ABB RobotStudio station: RoboX0_20211129-155304.rsstn

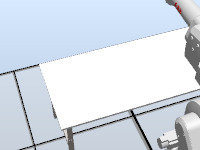
Station RoboX0 (saved by RobotStudio 21.3.9648.0)
Controller IRB1600_10_145, task T_ROB1: task frame (RAPID world) sits at (0, 0, 520) mm in the station
Controller IRB1600_10_145
  mechanical unit ROB_1: IRB1600_10_145__01_2, 6 joints, base frame (0, 0, 0) mm
Layout (positions relative to the parent item):
  - IRB1600_10_145__01_2 [mechanism, from Robots\IRB1600_10_145_G_01.rslib] at (0, 0, 520) mm; joint values [0, 0, 0, 0, 0.5236, 0] (rad or m)
  - подставка [part, from Libraries\box.rslib]
  - Стол сборка_4 [part, from Libraries\table.rslib] at (975, 0, 0) mm, rotated rx 0 ry 0 rz 90 deg
  - Frame_1 [frame] at (-300, -500, 0) mm
